% RSLogix 500 project ACIAIC.RSS, saved by version 9.00.00.04 %
PROJECT "UNTITLED"    % processor: Bul.1763 MicroLogix 1100 Series B %

PROGRAM FILES
  LAD 2   9 rungs

DATA FILES
  O0 OUTPUT  4 elements
  I1 INPUT  6 elements
  S2 STATUS  66 elements
  B3 BINARY  1 elements
  T4 TIMER  1 elements
  C5 COUNTER  1 elements
  R6 CONTROL  1 elements
  N7 INTEGER  1 elements
  F8 FLOAT  1 elements
  ST9 STRINGS  4 elements

LADDER 2
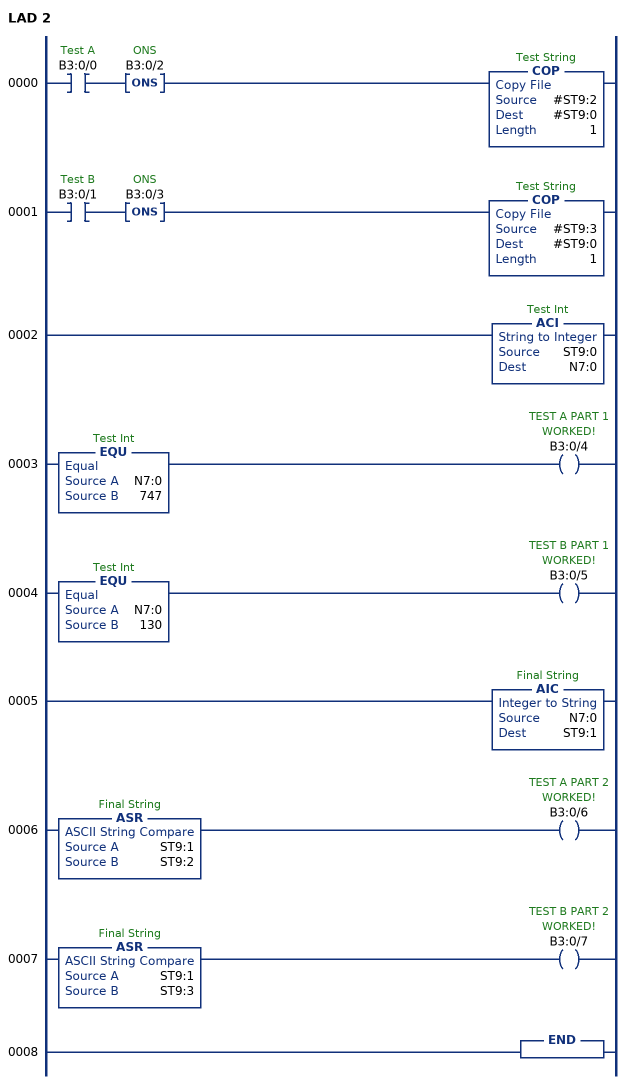
% Rung: 0 %
SOR XIC B3:0/0 ONS B3:0/2 COP #ST9:2 #ST9:0 1 EOR
%   B3:0/0  "Test A" %
%   B3:0/2  "ONS" %
%   ST9:2  "Test A Value" %
%   ST9:0  "Test String" %
% Rung: 1 %
SOR XIC B3:0/1 ONS B3:0/3 COP #ST9:3 #ST9:0 1 EOR
%   B3:0/1  "Test B" %
%   B3:0/3  "ONS" %
%   ST9:3  "Test B Value" %
%   ST9:0  "Test String" %
% Rung: 2 %
SOR ACI ST9:0 N7:0 EOR
%   ST9:0  "Test String" %
%   N7:0  "Test Int" %
% Rung: 3 %
SOR EQU N7:0 747 OTE B3:0/4 EOR
%   N7:0  "Test Int" %
%   B3:0/4  "TEST A PART 1 WORKED!" %
% Rung: 4 %
SOR EQU N7:0 130 OTE B3:0/5 EOR
%   N7:0  "Test Int" %
%   B3:0/5  "TEST B PART 1 WORKED!" %
% Rung: 5 %
SOR AIC N7:0 ST9:1 EOR
%   N7:0  "Test Int" %
%   ST9:1  "Final String" %
% Rung: 6 %
SOR ASR ST9:1 ST9:2 OTE B3:0/6 EOR
%   ST9:1  "Final String" %
%   ST9:2  "Test A Value" %
%   B3:0/6  "TEST A PART 2 WORKED!" %
% Rung: 7 %
SOR ASR ST9:1 ST9:3 OTE B3:0/7 EOR
%   ST9:1  "Final String" %
%   ST9:3  "Test B Value" %
%   B3:0/7  "TEST B PART 2 WORKED!" %
% Rung: 8 %
SOR END EOR

DATA TABLE (non-zero values as saved)
DATA ST9
% ST9:2 % "747"
% ST9:3 % "130"
